// TIA Portal V17 export
// export: Created 2021-12-03T08:13:11.225808Z, ExportSetting WithDefaults, DisplayName Totally Integrated Automation Portal, DisplayVersion V17, DisplayName TIA Portal Openness, DisplayVersion V17, DisplayName TIA Portal Version Control Interface, DisplayVersion V17, DisplayName STEP 7 Professional, DisplayVersion V17, DisplayName STEP 7 Safety, DisplayVersion V17, DisplayName WinCC Advanced, DisplayVersion V17
DATA_BLOCK "FDBI_EmStpButton"   // DB201, F_DB
VERSION : 0.1
// stored: AutoNumber false, InstanceOfName FFB_EmStpButton, InstanceOfType FB
"FFB_EmStpButton"
   // VAR
   //    P1 { S7_SetPoint := 'True'} : ESTOP1;
   //    P2 { S7_SetPoint := 'True'} : ESTOP1;
   //    P3 { S7_SetPoint := 'True'} : ESTOP1;
   //    AccCons { S7_SetPoint := 'True'} : ESTOP1;
   //    Dosimetr { S7_SetPoint := 'True'} : ESTOP1;
   // END_VAR
BEGIN
END_DATA_BLOCK
